Staubli VAL3: pLogger.pgx

public program pLogger()
  local joint jHere
  local point pHere
  local num nStart
  local num tEnd
begin
  //Definimos un punto inicial de logging sobre el que computar el tiempo relativo
  nStart=clock()
  //Quizas se pueda iniciar el logging ante una entrada digital que sincronice el laser tracker con el logging.
  while true
    tEnd = clock()-nStart
    sOutputMsgLog = "ts," +toString(".3", tEnd)
    jHere = herej()
    sOutputMsgLog = sOutputMsgLog + ",JOINTS," + toString(".3", jHere.j1) + "," + toString(".3", jHere.j2) + "," + toString(".3", jHere.j3) + "," + toString(".3", jHere.j4) + "," + toString(".3", jHere.j5) + "," + toString(".3", jHere.j6)
    pHere = here(tTool, world)
    sOutputMsgLog = sOutputMsgLog + ",CART,"
    sOutputMsgLog = sOutputMsgLog + toString(".3", pHere.trsf.x) + "," + toString(".3", pHere.trsf.y) + "," + toString(".3", pHere.trsf.z) + ","
    sOutputMsgLog = sOutputMsgLog + toString(".3", pHere.trsf.rx) + "," + toString(".3", pHere.trsf.ry) + "," + toString(".3", pHere.trsf.rz)
    sSio=sOutputMsgLog
    delay(0.02)
  endWhile
end
